VAR_GLOBAL CONSTANT
  MAX_PROCESS       : UINT := 5;
END_VAR
{attribute 'qualified_only'}
VAR_GLOBAL
  nDummy            : UINT;
END_VAR

(* stored: Version 1.1.0.1
   GVL GVL_APPLICATION: Id {b83de342-914f-4ad1-86ba-5efc40943708} *)
